TYPE ES_T6 :
STRUCT
		Alarm			:ES_ALARM;
	
		S1_rt			:R_TRIG;	
		S1_letto		:BOOL;
END_STRUCT
END_TYPE

(* stored: Version 1.1.0.1, ProductVersion 3.1.4022.6
   DUT ES_T6: Id {5b5759bc-efae-4be0-81e2-a4db95a2e4c0} *)
